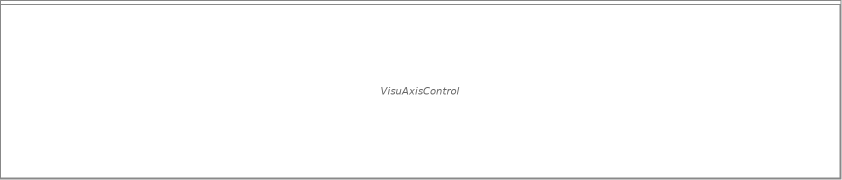
VISUALIZATION VisuAxisM1  // 842x180
    Frame (0,4 840x174)
        shows VisuAxisControl(sAxisName := sAxisM1_BName, stAxisVisu := stAxisM1_B)
END_VISUALIZATION

(* stored: Version 1.1.0.1, ProductVersion 3.1.4022.6
   Visu VisuAxisM1: Id {2bf8fb6b-d2f9-47ed-b6c7-8cddb38c7deb} *)
